{attribute addProperty BoxType "EL6080-0000-0018"}
{attribute addProperty Id "StatusAT %I*UINT162"}
{attribute addProperty CRC "2333909678"}
{attribute addProperty SizeInBites "16"}
{attribute addProperty SizeInBytes "2"}
TYPE Status_8B1CA2AE :
STRUCT
	{attribute addProperty Name "Status"}
	Status AT %I* : UINT;
END_STRUCT
END_TYPE

(* stored: Version 1.2.0.0, ProductVersion 3.1.4024.9
   DUT Status_8B1CA2AE: Id {bf6f9368-c3eb-4602-ae9c-5c1f83e92d0e} *)
